// TIA Portal V20 export
TYPE "IB_P01_02_03_out_64bytes_struct"
// stored: Access Published, Namespace Global
   STRUCT
      Run_mot_A : Bool;
      Run_mot_B : Bool;
      Reserved_1 : Bool;
      Reserved_2 : Bool;
      Reserved_3 : Bool;
      Reserved_4 : Bool;
      Reserved_5 : Bool;
      Reserved_6 : Bool;
      Speed_1_A : Bool;
      Speed_2_A : Bool;
      Speed_3_A : Bool;
      Speed_4_A : Bool;
      Speed_1_B : Bool;
      Speed_2_B : Bool;
      Speed_3_B : Bool;
      Speed_4_B : Bool;
      Acc_A : Bool;
      Dec_A : Bool;
      Acc_B : Bool;
      Dec_B : Bool;
      Dir_A : Bool;
      Dir_B : Bool;
      Ack_err_A : Bool;
      Ack_err_B : Bool;
      Digital_out1 : Bool;   // NA for IB-P03
      Digital_out2 : Bool;   // NA for IB-P03
      Digital_out3 : Bool;   // NA for IB-P03
      Digital_out4 : Bool;   // NA for IB-P03
      Reserved_7 : Bool;
      Reserved_8 : Bool;
      Reserved_9 : Bool;
      Reserved_10 : Bool;
      Register_Low_D800 : Byte;
      Register_High_D800 : Byte;
      Register_Low_D801 : Byte;
      Register_High_D801 : Byte;
      Register_Low_D802 : Byte;
      Register_High_D802 : Byte;
      Register_Low_D803 : Byte;
      Register_High_D803 : Byte;
      Register_Low_D804 : Byte;
      Register_High_D804 : Byte;
      Register_Low_D805 : Byte;
      Register_High_D805 : Byte;
      Register_Low_D806 : Byte;
      Register_High_D806 : Byte;
      Register_Low_D807 : Byte;
      Register_High_D807 : Byte;
      Register_Low_D808 : Byte;
      Register_High_D808 : Byte;
      Register_Low_D809 : Byte;
      Register_High_D809 : Byte;
      Register_Low_D810 : Byte;
      Register_High_D810 : Byte;
      Register_Low_D811 : Byte;
      Register_High_D811 : Byte;
      Register_Low_D812 : Byte;
      Register_High_D812 : Byte;
      Register_Low_D813 : Byte;
      Register_High_D813 : Byte;
      Register_Low_D814 : Byte;
      Register_High_D814 : Byte;
      Register_Low_D815 : Byte;
      Register_High_D815 : Byte;
      Output_stop : Byte;
      Led_JAM_A : Bool;
      Led_JAM_B : Bool;
      Led_soft1_A : Bool;
      Led_soft1_B : Bool;
      Led_soft2_A : Bool;
      Led_soft2_B : Bool;
      Reserved_11 : Bool;
      Reserved_12 : Bool;
      Reserved_13 : Array[0..25] of Byte;
   END_STRUCT;
END_TYPE
